(* IEC 61131-3 sources: eCockpitGit/test_project/src/%PLC%PLCTest2/%PLOG%Plc Logic/%APP%APP1_Test/%F%NormalFolder/%GVL%GVL_test_1/%F%GVLFolder/%PRO%PropAlop, 1 file *)

(* ---- %GETSET%Set.st ---- *)
VAR
	temp2:BOOL;
END_VAR

(*%!%__DELIMITER__%!%*)
variablssss		:=		temp2 AND PropAlop;
